(* This function is for the Cold Cathode MKS 500. 

If connected to Beckhoff EP boxes. Set the EP bit to TRUE, this is necessary for the 
IMG401-to-EP box interface because the EP boxes do not natively support the 5v IO 
signals on the gauge.

This function provides ILK and Set Point Protection for the hot Cathode.
*)

FUNCTION_BLOCK FB_IMG401 EXTENDS FB_GaugeBase
VAR_IN_OUT
		
END_VAR
VAR_INPUT
	PG	:	ST_VG;
	tRecoverDelay:TIME:=T#600S; (*Delay Time after the first cycle to start the device. Default is 600S*)
END_VAR
VAR_OUTPUT
{attribute 'pytmc' := '
    pv: 
	'}
	IG : ST_VG;
END_VAR
VAR
	rV : REAL;
	GaugeTurnOnTmr : TON;
	tStartupTimer:TON;
	iTermBits: UINT := 30518 ; // The terminal's maximum value in bits
	(*IOs to be linked*)
	/// Controls and I/Os
	i_iPRESS_R AT %I* :INT; // input Pressure // Link to analog Input
	q_xHV_DIS AT %Q* : BOOL; // Enable High Voltage when True // 'TcLinkTo' (EP2624) ^Output
	// only for EL and ES terminal
	i_xHV_ON AT %I*	: BOOL; //  True when High Voltage is on  // 'TcLinkTo' (EL1084) ^Input
//	i_xDisc_Active AT %I* : BOOL;// Discharge Current Active // 'TcLinkTo' (EL1124) ^Input
	binit:BOOL:=TRUE;
END_VAR

VAR CONSTANT
	vBase : REAL := 1.0;
	vDisconnected : REAL:= 0.001; //shift from 0 to eliminate single noise effect
	vTorr : REAL := 10; 
	vGaugeOff: REAL := 10;
	//vNoDischarge: REAL := 9.3;
	rMinPressure: REAL := 1E-10;
	cDefaultPressure : REAL := 0;
	rDeadband : REAL :=1.0;
END_VAR

VAR PERSISTENT
	bWasOn : BOOL;
	bAutoRecover:BOOL;
	bAutoRecoverWrite:BOOL;
END_VAR

(*Startup time*)
IF (bInit) THEN
	tStartupTimer.IN:=TRUE;
	bInit :=FALSE;
END_IF
tStartupTimer(PT:=T#3S);

If (iTermBits=0) THEN iTermBits := 32767;END_IF
rV := 10*INT_TO_REAL(IG.i_iPRESS_R)/iTermBits;


(* 401 Logarithmic Output Conversion, factory default configuration 
   EL3174, EL3174-xxxx iTermbits 30518, 10V
*)
If (iTermBits=0) THEN iTermBits := 30518;END_IF
rV := 10*INT_TO_REAL(IG.i_iPRESS_R)/iTermBits;

(* Set Guage State based on the Analog voltage*)

IF rV <= vDisconnected AND IG.i_xHV_ON and IG.q_xHV_DIS THEN
	IG.eState := ValidLo;
	IG.rPRESS := rMinPressure;
ELSIF rV <= vDisconnected AND NOT IG.i_xHV_ON and NOT IG.q_xHV_DIS THEN
	IG.eState := Off;
	IG.rPRESS := cDefaultPressure;
ELSIF rV <= vDisconnected AND Not IG.i_xHV_ON and IG.q_xHV_DIS THEN
	IG.eState := GaugeDisconnected;
	IG.rPRESS := cDefaultPressure;
ELSIF rV > vDisconnected AND rV < (vGaugeOff -rDeadband) AND IG.i_xHV_ON and IG.q_xHV_DIS THEN
	IG.eState := Valid;
	IG.rPRESS := LREAL_TO_REAL(EXPT(10,((rV*vBase)- vTorr)));
ELSIF rV >= (vGaugeOff -rDeadband) AND NOT IG.q_xHV_DIS THEN
	IG.eState := Off;
	IG.rPRESS := cDefaultPressure;
ELSE
	IG.eState := OoR;
	IG.rPRESS := cDefaultPressure;
END_IF



(* Ion Gauge Protection Functions *)
(* If the PG pressure is greater than the VG.PRO_SP then the gauge is disabled *)
(* If the PG pressure is less than the VG.PRO_SP then the gauge is enabled *)
(* This FB also implements some hysteresis so the gauge doesn't have rapid power cycling while near the turn on boundary *)


IF PG.rPRESS <= IG.rPRO_SP AND PG.xPRESS_OK THEN
	IG.q_xHV_DIS := IG.xHV_SW;
	IG.xILKOk := TRUE;
ELSIF IG.q_xHV_DIS THEN
	IF IG.rPRESS > (IG.rPRO_SP + IG.rHYS_PR)  OR PG.rPRESS > (IG.rPRO_SP + IG.rHYS_PR) THEN
		IG.q_xHV_DIS := FALSE;
		IG.xHV_SW := FALSE;
	END_IF
ELSE
	IG.q_xHV_DIS := FALSE;
	IG.xHV_SW := FALSE;
	IG.xILKOk := FALSE;
END_IF

(* Pressure gauge OK checks *)

GaugeTurnOnTmr(IN:=IG.q_xHV_DIS, PT:=T#10S, Q=>IG.xTurnOnTime);

//Backwards compatibility
IG.xPRESS_OK := (IG.eState = Valid) OR IG.xBAKEOUT;

(* Setpoint evaluation *)
IG.xAT_VAC := (IG.xPRESS_OK AND (IG.rPRESS < IG.rVAC_SP)) OR IG.xBAKEOUT AND (IG.eState = Valid) ;

ACT_Logger();
(*Soft IO Linking*)
// check ethercat Diagnostics
IO();
(*Load or save the persistent variables*)
ACT_Persistent();
(*Run Auto Recovery*)
ACT_Recover();

ACTION ACT_Logger:
// ILK logger
IF (IG.xLog) THEN
	IF NOT IG.xILKOk AND IG.q_xHV_DIS THEN
			fbLogger(sMsg:='Lost external interlock while gauge was on.', eSevr:=TcEventSeverity.Critical);  	
	END_IF
	
	
	// Log Action
	tAction(CLK:=   IG.xHV_SW);
	IF tAction.Q THEN fbLogger(sMsg:='Ion gauge commanded to switch on', eSevr:=TcEventSeverity.Info); END_IF
	
	
	
	//STATE Logger  
	tState(CLK:=  ePrevState <> IG.eState);
	IF ePrevState <> IG.eState THEN
		  CASE IG.eState OF
			ValidHi:
				fbLogger(sMsg:='Gauge pressure valid high.', eSevr:=TcEventSeverity.Info);
			ValidLo:
				fbLogger(sMsg:='Gauge pressure valid low.', eSevr:=TcEventSeverity.Info);
			Valid:
				fbLogger(sMsg:='Gauge pressure valid.', eSevr:=TcEventSeverity.Info);
			GaugeDisconnected:
				fbLogger(sMsg:='Gauge Disconnected.', eSevr:=TcEventSeverity.Critical);
			PressInvalid:
				fbLogger(sMsg:='Gauge pressure invalid.', eSevr:=TcEventSeverity.Warning);
			OoR:
				fbLogger(sMsg:='Gauge pressure out of range.', eSevr:=TcEventSeverity.Warning);
			Starting:
				fbLogger(sMsg:='Gauge starting.', eSevr:=TcEventSeverity.Info);
		  END_CASE
		  ePrevState := IG.eState;  
		  stateTimer.IN := TRUE;
	  END_IF
END_IF
END_ACTION

ACTION ACT_Persistent:
(*On first PLC pass, load the persistent value into the structrue variable*)
IF (SUPER^.bRestorePersistentData) THEN
	SUPER^.bRestorePersistentData	:= FALSE;
	IF ( rVAC_SP <> 0) THEN
		IG.rVAC_SP := rVAC_SP;
	END_IF;
	IF ( rPRO_SP <> 0) THEN
		IG.rPRO_SP := rPRO_SP;
	END_IF;
	IF ( rHYS_PR <> 0) THEN
		IG.rHYS_PR := rHYS_PR;
	END_IF;
	IF ( bAutoRecoverWrite) THEN
		IG.xAutoOn := bAutoRecover;
	END_IF;
END_IF
(*Check if a new value has been written in the structure variable copy it to the persistent variable*)
IF NOT (IG.rVAC_SP = rVAC_SP)  THEN
	rVAC_SP := IG.rVAC_SP;
END_IF;

IF NOT (IG.rPRO_SP = rPRO_SP) THEN
	rPRO_SP:= IG.rPRO_SP;
END_IF;

IF NOT (IG.rHYS_PR = rHYS_PR) THEN
	rHYS_PR:= IG.rHYS_PR;
END_IF;

IF NOT(bAutoRecoverWrite) OR NOT (bAutoRecover = IG.xAutoOn) THEN
	bAutoRecover := IG.xAutoOn;
	bAutoRecoverWrite := TRUE;
END_IF;
stateTimer(PT:=T#10S);
IF (stateTimer.Q) THEN
	bWasOn := (IG.eState >=Valid );
	stateTimer.IN := FALSE;
	fbWritePersistentData(NETID:='', PORT:=851, START:=TRUE, TMOUT:=T#1s );
END_IF;
END_ACTION

ACTION ACT_Recover:
fbGetCurTaskIdx();
IF (TwinCAT_SystemInfoVarList._TaskInfo[fbGetCurTaskIdx.index].FirstCycle) THEN
	tRecover.IN := TRUE;
END_IF
tRecover(IN:= , PT:=tRecoverDelay);
IF NOT(bAutoRecoverWrite) OR (tRecover.Q AND bAutoRecover ) THEN
	This^.M_Recover();
	tRecover.IN := FALSE;
END_IF
END_ACTION

ACTION IO:
(*soft link inputs*)
IG.i_iPRESS_R:=	i_iPRESS_R; 
IG.i_xHV_ON:= i_xHV_ON;
//IG.i_xDisc_Active:=i_xDisc_Active; 
(*soft link outputs*)
q_xHV_DIS := IG.q_xHV_DIS;

IG.sPath := sPath;
IG.iAutoOnTimer:= TIME_TO_INT(tRecover.PT);
END_ACTION

METHOD M_HVE : BOOL
VAR_INPUT
		enable:bool; // set to true to enable, false to disable;
END_VAR
this^.IG.xHV_SW:= enable;
END_METHOD

METHOD M_Recover : BOOL
VAR_INPUT
END_VAR
This^.M_HVE(This^.bWasOn);
M_Recover := bWasOn;
IF (bWasOn) THEN fbLogger(sMsg:='Auto Recovery Initiated.', eSevr:=TcEventSeverity.Info); END_IF;
END_METHOD

METHOD M_SetBits : BOOL
VAR_INPUT
	TermBits : UINT; // The terminal's maximum value in bits
END_VAR
This^.iTermBits := TermBits;
END_METHOD

END_FUNCTION_BLOCK

(* stored: Version 1.1.0.1, ProductVersion 3.1.4022.18
   POU FB_IMG401: Id {4a2fc267-eb2d-4ea0-9303-08a3354738d4}, SpecialFunc None
   Action ACT_Logger: Id {32bd2498-b785-470b-9d53-5fe2d5a7230c}
   Action ACT_Persistent: Id {19b99cce-686e-4553-a919-0f2d44f7d372}
   Action ACT_Recover: Id {1692d52d-07c8-44ef-8ca5-dd37315ae382}
   Action IO: Id {60cbf541-8efd-4b0a-8dbe-ac577a24b43e}
   Method M_HVE: Id {f2664a00-2f21-407e-9b83-88176d4d07a8}
   Method M_Recover: Id {34bdef07-51a5-4d00-b35d-f4abd6e58476}
   Method M_SetBits: Id {95269875-3fb6-4279-ba33-8df59a3308b4} *)
